{attribute 'qualified_only'}
{attribute 'strict'}
TYPE MsgLevel :
(
	Error	:= 4,
	Alarm	:= 2,
	Info	:= 1,
	None	:= 0
	
)INT;
END_TYPE

(* stored: Version 1.1.0.1, ProductVersion 3.1.4026.13
   DUT MsgLevel: Id {6741b6ff-79cc-4e2e-a47c-b5b77b5959b1} *)
